TYPE ST_TransportControl_Outputs :
(**************************************************************************************
 * 	Application		:	BoxControl Framework
 *	Revision		:	$Revision: 404529 $
 *	Revision date	:	$Date: 2018-04-23 08:21:38 +0200 (Mo., 23 Apr 2018) $
 *	Last changed by	:	$Author: b7bolm $
 *	URL				:	$URL: http://almscdc.swisslog.com/repo/SWPD/Development/BoxControlFramework/20_Release/trunk/01_Software/BCF/BCF/JumpStart/20_Product/10_App/12_E_Functions/10_Lib/10_Conv/10_Functions/01_DUTs/ST_TransportControl_Outputs.TcDUT $
 *
 *	Purpose			:	Transport control outputs
 *
 * ------------------------------------------------------------------------------------
 *	Copyright Swisslog [IP AG], Switzerland. All rights reserved.
 * 
 * ------------------------------------------------------------------------------------
 *	
 * 	Revision History: 
 *
 * 	VERSION			DATE			INITIALS			DESCRIPTION
 *	0.1				01.01.2001		swl					Example 
 *
 **************************************************************************************)	
STRUCT
	DriveRun   				 : BOOL; // Run signal for drive
	DriveTakeoverRun		 : BOOL; // Run signal for drive takeover
	DriveHandoverRun		 : BOOL; // Run signal for drive handover
	RequestPrevTransportData : BOOL; // Request previous transport data
	RequestNextTransportData : BOOL; // Request next transport data
	DeletePrevTransportData	 : BOOL; // Delete previous transport data
	DeleteNextTransportData  : BOOL; // Delete next transport data
	DistanceToZoneEnd		 : UINT; // Distance TU leading edge to zone end [mm]	
END_STRUCT
END_TYPE

(* stored: Version 1.1.0.1, ProductVersion 3.1.4022.12
   DUT ST_TransportControl_Outputs: Id {1a3f2353-1290-42e4-b46a-0bb8d37ce2ae} *)
